// TIA Portal project "Automated Curtain Control" (V17)
// Automated Curtain Control
// When the OPEN button is pressed, the curtains should open and remain open for 30 sec before closing automatically. If OPEN button is pressed again, the curtains will remain open for 30 sec more.

(* hardware
DEVICE "S7-1200 station_1"  S7-1200 Station
   slot 0: "Rack_0"  S7-1200 Rack  Rack  V1.0
   slot 1: "PLC_1"  CPU 1215C AC/DC/Rly  6ES7 215-1BG40-0XB0  V4.5
*)

// ===== PLC "PLC_1"  CPU 1215C AC/DC/Rly =====

VAR_GLOBAL   // PLC tag table "Default tag table"
   "pb open" AT %I0.0 : Bool;
   "curtain" AT %Q0.0 : Bool;
   "Tag_1" AT %M0.0 : Bool;
   "Tag_2" AT %M0.1 : Bool;
   "Tag_3" AT %M0.2 : Bool;
   "Tag_4" AT %M0.3 : Bool;
   "Tag_5" AT %M0.4 : Bool;
END_VAR

// folder: System blocks/Program resources

DATA_BLOCK "IEC_Timer_0_DB"   // DB1
{ S7_Optimized_Access := 'TRUE' }
AUTHOR : Simatic
FAMILY : IEC
NAME : IEC_TMR
VERSION : 1.0
// stored: InstanceOfName IEC_TIMER
"IEC_TIMER"
BEGIN
END_DATA_BLOCK

DATA_BLOCK "IEC_Timer_0_DB_1"   // DB2
{ S7_Optimized_Access := 'TRUE' }
AUTHOR : Simatic
FAMILY : IEC
NAME : IEC_TMR
VERSION : 1.0
// stored: InstanceOfName IEC_TIMER
"IEC_TIMER"
BEGIN
END_DATA_BLOCK

// folder: (top level)

ORGANIZATION_BLOCK "Main"   // OB1, LAD, ProgramCycle
TITLE = "Main Program Sweep (Cycle)"
{ S7_Optimized_Access := 'TRUE' }
VERSION : 0.1
   VAR_INPUT
      Initial_Call : Bool;   // Initial call of this OB
      Remanence : Bool;   // =True, if remanent data are available
   END_VAR
BEGIN

REGION Network 1
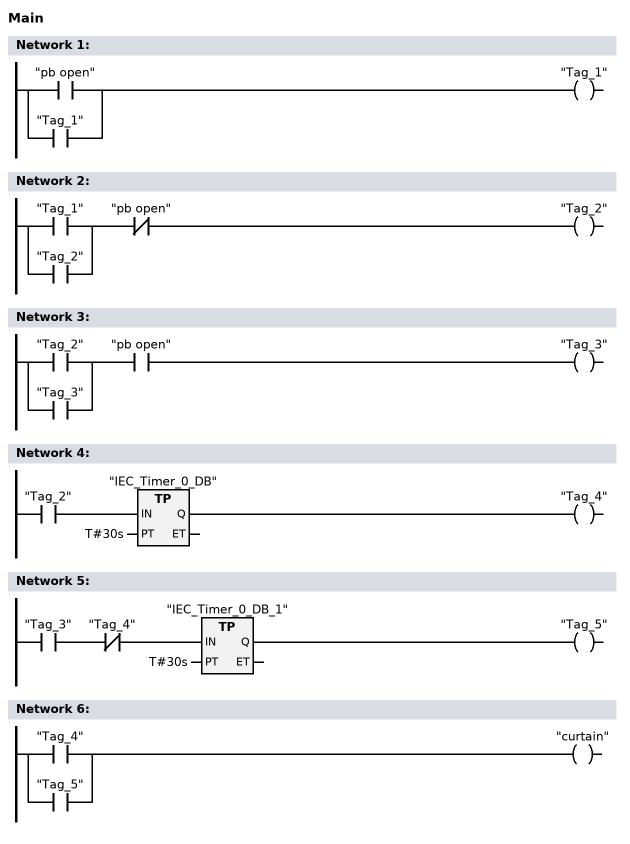
   RUNG wire#powerrail
      Contact( "pb open" )
      wire#w1
      Coil( "Tag_1" )
   END_RUNG
   RUNG wire#powerrail
      Contact( "Tag_1" )
   END_RUNG wire#w1
   // the same network as SCL:
   "Tag_1" := "pb open" OR "Tag_1";
END_REGION

REGION Network 2
   RUNG wire#powerrail
      Contact( "Tag_1" )
      wire#w1
      I_Contact( "pb open" )
      Coil( "Tag_2" )
   END_RUNG
   RUNG wire#powerrail
      Contact( "Tag_2" )
   END_RUNG wire#w1
   // the same network as SCL:
   "Tag_2" := ("Tag_1" OR "Tag_2") AND NOT "pb open";
END_REGION

REGION Network 3
   RUNG wire#powerrail
      Contact( "Tag_2" )
      wire#w1
      Contact( "pb open" )
      Coil( "Tag_3" )
   END_RUNG
   RUNG wire#powerrail
      Contact( "Tag_3" )
   END_RUNG wire#w1
   // the same network as SCL:
   "Tag_3" := ("Tag_2" OR "Tag_3") AND "pb open";
END_REGION

REGION Network 4
   "IEC_Timer_0_DB".TP(IN := "Tag_2", PT := T#30s);
   "Tag_4" := "IEC_Timer_0_DB".Q;
END_REGION

REGION Network 5
   "IEC_Timer_0_DB_1".TP(IN := "Tag_3" AND NOT "Tag_4", PT := T#30s);
   "Tag_5" := "IEC_Timer_0_DB_1".Q;
END_REGION

REGION Network 6
   RUNG wire#powerrail
      Contact( "Tag_4" )
      wire#w1
      Coil( "curtain" )
   END_RUNG
   RUNG wire#powerrail
      Contact( "Tag_5" )
   END_RUNG wire#w1
   // the same network as SCL:
   "curtain" := "Tag_4" OR "Tag_5";
END_REGION
END_ORGANIZATION_BLOCK